FUNCTION_BLOCK FB_Control
VAR_INPUT
	button1: BOOL;
	ProcessDone: BOOL;
	StopDone: BOOL;
END_VAR
VAR_OUTPUT
	position: LREAL;
	ProgEx: BOOL;
	StopState: BOOL;
END_VAR
VAR
	nState: INT;
	TON1: TON;
	TON2: TON;
	TON3: TON;
	R_TRIG1: R_TRIG;
	F_TRIG1: F_TRIG;
END_VAR
VAR_IN_OUT
	
	
END_VAR



CASE nState OF
0:
	
	IF button1 THEN
		StopState:=FALSE;
		nState:=10;
	END_IF
10:
	nState:=15;
	position:=30000;
	progEx:=TRUE;

15:
	
IF ProcessDone THEN
	TON1(IN:=TRUE, PT:=T#1S , Q=> , ET=> );
	IF TON1.Q THEN
		nState:=19;
		TON1(IN:=FALSE);

	END_IF
END_IF

19:
	ProgEx:=FALSE;
	nState:=20;

20:
	position:=20000;
	nState	:=25;
	progEx	:=TRUE;


25:
IF ProcessDone THEN
		TON2(IN:=TRUE, PT:=T#4S , Q=> , ET=> );
	IF TON2.Q THEN
		nState:=26;
		TON2(IN:=FALSE);
	END_IF
END_IF

26:
	ProgEx:=FALSE;
	nState:=30;

30:
	position:=0;
	nState:=35;
	progEx:=TRUE;

35:
IF ProcessDone THEN
		TON3(IN:=TRUE, PT:=T#2S , Q=> , ET=> );
	IF TON3.Q THEN
		nState:=36;
		TON3(IN:=FALSE);
	END_IF
END_IF
36:
	
	ProgEx:=FALSE;
	nState:=0;

100:
	StopState:=TRUE;
	IF StopDone THEN
		nState:=0;
		TON1(IN:=FALSE);
		TON2(IN:=FALSE);
		TON3(IN:=FALSE);
		ProgEx:=FALSE;
		StopState:=FALSE;

END_IF
END_CASE
F_TRIG1(CLK:=button1 , Q=> );

IF F_TRIG1.Q THEN
	nState:=100;
END_IF

END_FUNCTION_BLOCK

(* stored: Version 1.1.0.1, ProductVersion 3.1.4022.16
   POU FB_Control: Id {e52de16d-7a51-46f2-8ee6-cf9e07effbca}, SpecialFunc None *)
